Fanuc KAREL source: kb00065.KL

-- PROVISIONAL review KL for V940-1; original PC SHA256 993653beb8e3268b994b8eb5ea8a1cfb17206a5d12a277046cbf4870640ffe00
-- Incomplete behavior may be omitted. Consult companion uncertainty JSON. Do not deploy.
PROGRAM KB00065
%NOLOCKGROUP
BEGIN
  -- V9_ZERO_TABLE_METADATA_HINT layout=0002_ascii; no indexed target words; source/name/runtime held
  -- UNRESOLVED_PC offsets 5-14; opcodes 3F,75
  -- UNRESOLVED_PC offsets 19-26; opcodes 9D,23
  -- UNRESOLVED_PC offsets 31-38; opcodes 9D,23
  -- UNRESOLVED_PC offsets 43-52; opcodes 3F,75
  -- UNRESOLVED_PC offsets 57-66; opcodes 3F,75
  -- UNRESOLVED_PC offsets 71-78; opcodes 9D,23
  -- UNRESOLVED_PC offsets 83-90; opcodes 9D,23
  -- UNRESOLVED_PC offsets 95-102; opcodes 9D,23
  -- UNRESOLVED_PC offsets 107-165; opcodes 27,22,2A,22,22,22,2A,22,2A,22,22,22,31
  -- UNRESOLVED_PC offsets 170-174; opcodes 7F
END KB00065
